{attribute 'linkalways'} 
{attribute 'no_explicit_call' := 'This FB is a CLASS and must be accessed using methods or properties'}
{attribute 'enable_dynamic_creation'}
FUNCTION_BLOCK Node_F_VN_ImageMedianExp EXTENDS VisionNode
VAR
    ipSrcImage : _ITcVnImage;
    aMedian : _TcVnVector4_LREAL;
    ipMask : _ITcVnImage;
    hrPrev : _HRESULT(S_OK);
	hresult : _HRESULT(S_OK);
END_VAR

METHOD PUBLIC  Clone : I_Node
VAR
	pNode : POINTER TO Node_F_VN_ImageMedianExp;
END_VAR
pNode := __NEW(Node_F_VN_ImageMedianExp);
Clone := pNode^;
END_METHOD

METHOD FB_init : BOOL
VAR_INPUT
	bInitRetains : BOOL; // if TRUE, the retain variables are initialized (warm start / cold start)
	bInCopyCode : BOOL;  // if TRUE, the instance afterwards gets moved into the copy code (online change)
END_VAR
AddInput('ipSrcImage', ipSrcImage);
AddInput('ipMask', ipMask);
AddInput('hrPrev', hrPrev);
AddOutput('aMedian', aMedian);
AddOutput('hresult', hresult);
END_METHOD

METHOD PROTECTED  OnExecute : HRESULT
hresult.Value := F_VN_ImageMedianExp(
	ipSrcImage := ipSrcImage.Value,
    aMedian := aMedian.Value,
    ipMask := ipMask.Value,
	hrPrev:= hrPrev.Value);
END_METHOD

METHOD PUBLIC PreExecutionCheck
VAR_INPUT
	Check : I_PreExecutionChecks;
END_VAR
Check.IsTrue(ipSrcImage.IsValid, 'ipSrcImage must contain an image');
Check.IsTrue((ipSrcImage.HasChannelCount(1) OR
              ipSrcImage.HasChannelCount(2) OR
              ipSrcImage.HasChannelCount(3) OR
              ipSrcImage.HasChannelCount(4)), 'ipSrcImage must contain 1, 2, 3 or 4 channels');

Check.IsTrue(ipMask.IsValid, 'ipMask must contain an image');
Check.IsTrue(ipMask.HasChannelCount(1), 'ipMask must have 1 channel');
Check.IsTrue(ipMask.IsPixelDepth(8), 'ipMask must have 8 bit pixel depth');
Check.IsTrue(IsImage1SizeEqualToImage2Size(ipMask.Value, ipSrcImage.Value), 'ipMask must be the same size as ipSrcImage');
END_METHOD

END_FUNCTION_BLOCK

(* stored: Version 1.1.0.1, ProductVersion 3.1.4024.13
   POU Node_F_VN_ImageMedianExp: Id {aa355913-f639-05c3-2b1f-7a176130e39f}, SpecialFunc None
   Folder Constructor: Id {fdf04f19-3ef1-01fe-1d85-b66a2e2aebc7}
   Method Clone: Id {00c33831-e7d9-0c07-2748-b10bd5f3c9fe}
   Method FB_init: Id {c226722d-2221-093f-10ea-494a21273ba9}
   Method OnExecute: Id {ca68f122-298f-006e-3104-ccc434bc3de1}
   Method PreExecutionCheck: Id {e69cedd3-9270-0fc4-23fb-77b63ef6b310} *)
